Yaskawa INFORM job: DPRINT3D18.JBI

/JOB
//NAME DPRINT3D18
//POS
///NPOS 625,0,0,0,0,0
///TOOL 9
///POSTYPE PULSE
///PULSE
C00000=36096,32575,-120643,81709,-123035,-81395,0
C00001=36425,32776,-120243,81467,-123331,-81351,0
C00002=34958,34612,-116515,83246,-122769,-80325,0
C00003=34636,34416,-116909,83476,-122474,-80372,0
C00004=34349,34800,-116126,83824,-122361,-80159,0
C00005=35252,35359,-115002,83189,-123196,-80022,0
C00006=35016,35676,-114352,83478,-123103,-79844,0
C00007=35485,35977,-113744,83156,-123545,-79768,0
C00008=35668,35733,-114245,82930,-123616,-79906,0
C00009=36231,35313,-115109,82324,-123921,-80177,0
C00010=38030,32425,-120969,79919,-124380,-81738,0
C00011=40285,30090,-125653,77187,-125198,-83094,0
C00012=40286,30038,-125645,77208,-125225,-83061,0
C00013=36418,35187,-115263,82157,-124059,-80209,0
C00014=41098,30074,-125584,76447,-125785,-83178,0
C00015=40091,29408,-126885,77224,-124886,-83293,0
C00016=37256,32373,-120954,80642,-123847,-81594,0
C00017=37581,32580,-120545,80403,-124142,-81550,0
C00018=35772,34768,-116105,82607,-123455,-80311,0
C00019=36340,35136,-115366,82211,-123986,-80222,0
C00020=35723,35614,-114384,82881,-123656,-79916,0
C00021=36597,36197,-113208,82288,-124488,-79769,0
C00022=47213,22031,-141100,88472,-114439,-84668,0
C00023=39961,28432,-128797,77096,-124480,-83674,0
C00024=36097,32526,-120634,81728,-123056,-81363,0
C00025=36425,32727,-120235,81485,-123353,-81319,0
C00026=34959,34565,-116507,83263,-122787,-80294,0
C00027=34636,34368,-116901,83493,-122492,-80341,0
C00028=34350,34753,-116118,83841,-122379,-80128,0
C00029=35253,35312,-114994,83206,-123215,-79992,0
C00030=35016,35630,-114344,83496,-123122,-79813,0
C00031=35485,35931,-113736,83174,-123563,-79737,0
C00032=35669,35686,-114237,82948,-123634,-79875,0
C00033=36231,35266,-115101,82343,-123941,-80147,0
C00034=38031,32375,-120961,79938,-124402,-81706,0
C00035=40286,30038,-125645,77208,-125225,-83061,0
C00036=40286,29986,-125636,77229,-125250,-83028,0
C00037=36419,35140,-115255,82176,-124079,-80178,0
C00038=41098,30022,-125576,76469,-125813,-83145,0
C00039=40091,29355,-126877,77245,-124912,-83260,0
C00040=37256,32324,-120946,80661,-123870,-81562,0
C00041=37581,32531,-120536,80423,-124165,-81518,0
C00042=35772,34721,-116097,82625,-123474,-80280,0
C00043=36341,35089,-115358,82229,-124005,-80191,0
C00044=35723,35568,-114376,82899,-123674,-79885,0
C00045=36598,36150,-113200,82307,-124508,-79739,0
C00046=47214,21968,-141090,88484,-114457,-84628,0
C00047=39961,28378,-128788,77117,-124508,-83641,0
C00048=36097,32476,-120626,81746,-123078,-81331,0
C00049=36425,32677,-120226,81504,-123373,-81287,0
C00050=34959,34517,-116499,83281,-122807,-80263,0
C00051=34636,34320,-116893,83511,-122511,-80310,0
C00052=34350,34705,-116110,83858,-122398,-80098,0
C00053=35253,35265,-114985,83224,-123233,-79961,0
C00054=35016,35583,-114335,83514,-123140,-79783,0
C00055=35485,35885,-113727,83192,-123581,-79707,0
C00056=35669,35640,-114229,82966,-123654,-79845,0
C00057=36231,35219,-115093,82361,-123961,-80116,0
C00058=38031,32326,-120953,79958,-124425,-81674,0
C00059=40286,29986,-125636,77229,-125250,-83028,0
C00060=40286,29934,-125628,77250,-125276,-82995,0
C00061=36419,35093,-115247,82194,-124100,-80148,0
C00062=41099,29970,-125567,76490,-125839,-83112,0
C00063=40092,29302,-126868,77266,-124938,-83226,0
C00064=37257,32274,-120938,80680,-123892,-81529,0
C00065=37581,32481,-120528,80442,-124187,-81486,0
C00066=35773,34674,-116088,82643,-123493,-80249,0
C00067=36341,35042,-115350,82248,-124025,-80160,0
C00068=35724,35521,-114368,82917,-123694,-79855,0
C00069=36598,36104,-113191,82326,-124527,-79708,0
C00070=47215,21905,-141081,88497,-114476,-84588,0
C00071=39961,28324,-128780,77137,-124535,-83607,0
C00072=36097,32426,-120618,81764,-123099,-81299,0
C00073=36426,32628,-120218,81522,-123395,-81255,0
C00074=34959,34470,-116490,83298,-122825,-80232,0
C00075=34637,34273,-116885,83528,-122530,-80279,0
C00076=34350,34658,-116101,83875,-122416,-80067,0
C00077=35253,35218,-114976,83242,-123252,-79930,0
C00078=35017,35536,-114327,83531,-123158,-79752,0
C00079=35486,35838,-113719,83210,-123600,-79676,0
C00080=35669,35593,-114221,82984,-123672,-79815,0
C00081=36232,35172,-115084,82379,-123980,-80086,0
C00082=38031,32276,-120944,79978,-124448,-81642,0
C00083=40286,29934,-125628,77250,-125276,-82995,0
C00084=40287,29882,-125619,77271,-125303,-82962,0
C00085=36419,35046,-115237,82213,-124119,-80117,0
C00086=41099,29918,-125559,76511,-125867,-83079,0
C00087=40092,29249,-126859,77287,-124965,-83193,0
C00088=37257,32224,-120929,80700,-123913,-81497,0
C00089=37582,32432,-120519,80461,-124209,-81454,0
C00090=35773,34626,-116080,82661,-123512,-80218,0
C00091=36341,34995,-115341,82266,-124046,-80130,0
C00092=35724,35475,-114359,82935,-123712,-79824,0
C00093=36598,36058,-113183,82344,-124545,-79678,0
C00094=47215,21842,-141070,88510,-114494,-84548,0
C00095=39962,28270,-128771,77158,-124562,-83572,0
C00096=36098,32377,-120608,81783,-123119,-81266,0
C00097=36426,32579,-120209,81541,-123416,-81223,0
C00098=34960,34422,-116482,83316,-122845,-80201,0
C00099=34637,34225,-116876,83545,-122548,-80247,0
C00100=34351,34611,-116092,83892,-122434,-80036,0
C00101=35254,35172,-114968,83259,-123270,-79899,0
C00102=35017,35490,-114319,83549,-123177,-79722,0
C00103=35486,35792,-113711,83228,-123618,-79646,0
C00104=35670,35547,-114212,83002,-123691,-79784,0
C00105=36232,35125,-115075,82398,-124000,-80055,0
C00106=38032,32226,-120936,79997,-124471,-81610,0
C00107=40287,29882,-125619,77271,-125303,-82962,0
C00108=40287,29829,-125610,77292,-125329,-82929,0
C00109=36419,34999,-115229,82231,-124139,-80087,0
C00110=41100,29866,-125550,76533,-125893,-83046,0
C00111=40093,29196,-126850,77308,-124991,-83160,0
C00112=37257,32175,-120920,80719,-123935,-81465,0
C00113=37582,32382,-120511,80480,-124232,-81422,0
C00114=35773,34579,-116072,82680,-123532,-80187,0
C00115=36342,34948,-115333,82285,-124065,-80099,0
C00116=35724,35428,-114351,82953,-123731,-79794,0
C00117=36599,36012,-113174,82363,-124565,-79648,0
C00118=47216,21778,-141061,88523,-114513,-84508,0
C00119=39962,28216,-128762,77179,-124589,-83539,0
C00120=36098,32328,-120600,81801,-123140,-81234,0
C00121=36427,32530,-120201,81559,-123437,-81191,0
C00122=34960,34375,-116474,83334,-122863,-80170,0
C00123=34638,34177,-116868,83563,-122567,-80217,0
C00124=34351,34564,-116084,83910,-122453,-80005,0
C00125=35254,35125,-114959,83277,-123289,-79868,0
C00126=35018,35444,-114310,83566,-123195,-79692,0
C00127=35487,35746,-113702,83246,-123636,-79615,0
C00128=35670,35500,-114204,83020,-123710,-79754,0
C00129=36232,35078,-115067,82416,-124019,-80024,0
C00130=38032,32177,-120927,80017,-124493,-81579,0
C00131=40287,29829,-125610,77292,-125329,-82929,0
C00132=40288,29777,-125600,77313,-125356,-82895,0
C00133=36420,34953,-115220,82250,-124158,-80056,0
C00134=41100,29814,-125541,76555,-125921,-83013,0
C00135=40093,29143,-126841,77329,-125019,-83126,0
C00136=37258,32125,-120912,80738,-123957,-81433,0
C00137=37583,32333,-120502,80500,-124254,-81390,0
C00138=35774,34532,-116062,82698,-123551,-80156,0
C00139=36342,34901,-115324,82303,-124085,-80068,0
C00140=35725,35382,-114342,82972,-123750,-79763,0
C00141=36599,35967,-113166,82382,-124585,-79617,0
C00142=47216,21715,-141051,88536,-114531,-84467,0
C00143=39963,28162,-128753,77200,-124617,-83504,0
C00144=36098,32278,-120591,81820,-123162,-81203,0
C00145=36427,32481,-120191,81578,-123458,-81160,0
C00146=34960,34327,-116465,83351,-122882,-80139,0
C00147=34638,34130,-116859,83580,-122586,-80185,0
C00148=34351,34516,-116075,83927,-122471,-79974,0
C00149=35254,35078,-114951,83295,-123308,-79838,0
C00150=35018,35397,-114302,83584,-123214,-79661,0
C00151=35487,35700,-113694,83264,-123655,-79585,0
C00152=35670,35454,-114195,83038,-123728,-79723,0
C00153=36233,35031,-115058,82435,-124039,-79993,0
C00154=38033,32127,-120919,80037,-124516,-81547,0
C00155=40288,29777,-125600,77313,-125356,-82895,0
C00156=40288,29725,-125592,77334,-125382,-82862,0
C00157=36420,34906,-115212,82268,-124178,-80025,0
C00158=41101,29762,-125531,76576,-125947,-82980,0
C00159=40093,29091,-126832,77350,-125045,-83092,0
C00160=37258,32076,-120903,80757,-123979,-81401,0
C00161=37583,32284,-120492,80519,-124275,-81358,0
C00162=35774,34485,-116053,82716,-123571,-80125,0
C00163=36342,34854,-115315,82322,-124104,-80037,0
C00164=35725,35335,-114333,82990,-123769,-79733,0
C00165=36599,35921,-113157,82400,-124603,-79587,0
C00166=47217,21652,-141040,88549,-114550,-84427,0
C00167=39963,28108,-128743,77221,-124644,-83470,0
C00168=36099,32229,-120582,81838,-123183,-81171,0
C00169=36427,32431,-120183,81597,-123479,-81128,0
C00170=34961,34280,-116457,83369,-122901,-80108,0
C00171=34638,34082,-116851,83598,-122605,-80154,0
C00172=34352,34469,-116067,83944,-122490,-79943,0
C00173=35254,35031,-114942,83313,-123326,-79807,0
C00174=35018,35351,-114293,83602,-123231,-79630,0
C00175=35487,35654,-113685,83282,-123673,-79555,0
C00176=35671,35407,-114186,83056,-123747,-79692,0
C00177=36233,34985,-115050,82453,-124058,-79962,0
C00178=38033,32078,-120910,80056,-124539,-81514,0
C00179=40288,29725,-125592,77334,-125382,-82862,0
C00180=40288,29673,-125583,77356,-125408,-82829,0
C00181=36421,34859,-115203,82287,-124197,-79994,0
C00182=41101,29710,-125522,76598,-125975,-82947,0
C00183=40094,29038,-126823,77371,-125072,-83059,0
C00184=37258,32026,-120893,80776,-124001,-81369,0
C00185=37583,32234,-120484,80539,-124297,-81326,0
C00186=35774,34438,-116045,82734,-123591,-80094,0
C00187=36342,34808,-115306,82341,-124124,-80007,0
C00188=35725,35289,-114325,83008,-123787,-79702,0
C00189=36600,35875,-113149,82419,-124622,-79557,0
C00190=47217,21590,-141030,88562,-114568,-84386,0
C00191=39963,28054,-128734,77242,-124671,-83436,0
C00192=36099,32180,-120574,81857,-123203,-81138,0
C00193=36428,32382,-120174,81615,-123500,-81096,0
C00194=34961,34233,-116447,83387,-122919,-80077,0
C00195=34639,34035,-116842,83615,-122623,-80123,0
C00196=34352,34422,-116058,83961,-122507,-79912,0
C00197=35255,34985,-114934,83331,-123345,-79776,0
C00198=35018,35304,-114284,83619,-123249,-79599,0
C00199=35487,35608,-113676,83300,-123692,-79524,0
C00200=35671,35361,-114178,83075,-123765,-79662,0
C00201=36233,34938,-115041,82472,-124078,-79932,0
C00202=38033,32028,-120900,80076,-124562,-81482,0
C00203=40288,29673,-125583,77356,-125408,-82829,0
C00204=40289,29621,-125574,77377,-125435,-82796,0
C00205=36421,34812,-115195,82306,-124217,-79963,0
C00206=41101,29658,-125513,76620,-126001,-82914,0
C00207=40094,28985,-126814,77392,-125098,-83025,0
C00208=37259,31977,-120884,80796,-124024,-81337,0
C00209=37584,32185,-120475,80558,-124320,-81294,0
C00210=35775,34391,-116036,82752,-123609,-80063,0
C00211=36343,34761,-115297,82359,-124143,-79976,0
C00212=35726,35243,-114316,83026,-123807,-79671,0
C00213=36600,35829,-113140,82438,-124641,-79526,0
C00214=47218,21527,-141020,88574,-114586,-84346,0
C00215=39964,28000,-128725,77264,-124698,-83402,0
C00216=36099,32130,-120565,81875,-123224,-81106,0
C00217=36428,32333,-120165,81634,-123522,-81064,0
C00218=34961,34186,-116438,83404,-122938,-80045,0
C00219=34639,33987,-116832,83633,-122641,-80092,0
C00220=34352,34375,-116049,83979,-122525,-79881,0
C00221=35255,34938,-114925,83349,-123363,-79745,0
C00222=35019,35258,-114275,83637,-123268,-79569,0
C00223=35488,35562,-113667,83318,-123710,-79494,0
C00224=35671,35315,-114169,83093,-123785,-79631,0
C00225=36234,34891,-115032,82490,-124096,-79901,0
C00226=38034,31979,-120891,80096,-124583,-81450,0
C00227=40289,29621,-125574,77377,-125435,-82796,0
C00228=40289,29570,-125564,77398,-125461,-82763,0
C00229=36421,34766,-115186,82324,-124236,-79932,0
C00230=41102,29606,-125504,76641,-126029,-82881,0
C00231=40095,28933,-126804,77413,-125125,-82991,0
C00232=35457,34141,-116430,82993,-123333,-80080,0
C00233=36343,34714,-115289,82378,-124163,-79944,0
C00234=35726,35196,-114307,83044,-123825,-79641,0
C00235=36600,35783,-113131,82457,-124660,-79496,0
C00236=47218,21464,-141009,88587,-114605,-84306,0
C00237=39964,27947,-128715,77285,-124726,-83367,0
C00238=34353,34328,-116041,83996,-122544,-79850,0
C00239=35256,34892,-114916,83367,-123383,-79715,0
C00240=35019,35212,-114266,83655,-123286,-79538,0
C00241=35488,35516,-113658,83336,-123728,-79463,0
C00242=35672,35269,-114160,83111,-123803,-79600,0
C00243=36234,34845,-115024,82509,-124116,-79870,0
C00244=36199,34122,-116480,82342,-123887,-80190,0
C00245=40289,29570,-125564,77398,-125461,-82763,0
C00246=40290,29518,-125554,77419,-125488,-82729,0
C00247=36422,34719,-115176,82343,-124256,-79902,0
C00248=41102,29554,-125495,76663,-126055,-82847,0
C00249=40095,28880,-126794,77435,-125151,-82958,0
C00250=35457,34094,-116421,83011,-123352,-80048,0
C00251=36344,34667,-115280,82397,-124182,-79914,0
C00252=35726,35150,-114298,83063,-123843,-79610,0
C00253=36601,35738,-113122,82475,-124680,-79466,0
C00254=47219,21401,-140999,88600,-114623,-84266,0
C00255=39965,27893,-128705,77306,-124753,-83333,0
C00256=34353,34281,-116031,84013,-122562,-79819,0
C00257=35256,34845,-114907,83385,-123401,-79684,0
C00258=35019,35166,-114257,83673,-123304,-79508,0
C00259=35488,35470,-113649,83354,-123747,-79433,0
C00260=35672,35223,-114151,83129,-123822,-79570,0
C00261=36234,34798,-115014,82527,-124135,-79839,0
C00262=36199,34074,-116470,82360,-123907,-80159,0
C00263=40290,29518,-125554,77419,-125488,-82729,0
C00264=40290,29466,-125545,77441,-125513,-82696,0
C00265=36422,34673,-115167,82362,-124275,-79871,0
C00266=41103,29503,-125485,76685,-126083,-82814,0
C00267=40095,28828,-126785,77456,-125178,-82924,0
C00268=35458,34047,-116413,83030,-123371,-80017,0
C00269=36344,34621,-115271,82415,-124202,-79883,0
C00270=35727,35104,-114289,83081,-123863,-79580,0
C00271=36601,35692,-113113,82494,-124698,-79435,0
C00272=47220,21338,-140988,88614,-114642,-84225,0
C00273=39965,27839,-128696,77327,-124780,-83299,0
C00274=34353,34234,-116022,84031,-122580,-79787,0
C00275=35256,34799,-114898,83403,-123419,-79653,0
C00276=35020,35120,-114248,83691,-123323,-79477,0
C00277=35489,35424,-113640,83372,-123766,-79402,0
C00278=35672,35177,-114142,83147,-123841,-79539,0
C00279=36235,34752,-115005,82546,-124155,-79809,0
C00280=36200,34027,-116461,82379,-123927,-80128,0
C00281=40290,29466,-125545,77441,-125513,-82696,0
C00282=40291,29414,-125536,77462,-125539,-82662,0
C00283=36422,34626,-115158,82381,-124295,-79839,0
C00284=41103,29451,-125475,76707,-126109,-82781,0
C00285=40096,28775,-126775,77477,-125205,-82891,0
C00286=35458,34000,-116403,83048,-123391,-79986,0
C00287=36344,34574,-115261,82434,-124221,-79852,0
C00288=35727,35058,-114280,83099,-123881,-79549,0
C00289=36601,35646,-113104,82513,-124718,-79405,0
C00290=47220,21276,-140977,88627,-114660,-84185,0
C00291=39966,27786,-128686,77349,-124807,-83265,0
C00292=34354,34187,-116013,84048,-122599,-79756,0
C00293=35256,34753,-114889,83421,-123438,-79622,0
C00294=35020,35074,-114239,83709,-123341,-79446,0
C00295=35489,35378,-113631,83390,-123785,-79371,0
C00296=35673,35131,-114133,83166,-123859,-79509,0
C00297=36235,34706,-114996,82565,-124174,-79778,0
C00298=36200,33980,-116452,82398,-123947,-80097,0
C00299=40291,29414,-125536,77462,-125539,-82662,0
C00300=40291,29363,-125526,77484,-125566,-82629,0
C00301=36423,34580,-115149,82400,-124314,-79809,0
C00302=41103,29399,-125466,76729,-126137,-82748,0
C00303=40096,28723,-126766,77498,-125232,-82857,0
C00304=35458,33953,-116393,83066,-123409,-79955,0
C00305=36345,34528,-115252,82453,-124241,-79821,0
C00306=35727,35012,-114270,83118,-123900,-79518,0
C00307=36602,35601,-113094,82532,-124737,-79374,0
C00308=47221,21213,-140967,88640,-114679,-84144,0
C00309=39966,27732,-128677,77370,-124835,-83231,0
C00310=34354,34140,-116004,84066,-122616,-79725,0
C00311=35257,34706,-114879,83439,-123456,-79591,0
C00312=35020,35028,-114230,83726,-123360,-79415,0
C00313=35489,35332,-113622,83408,-123803,-79341,0
C00314=35673,35084,-114123,83184,-123878,-79478,0
C00315=36235,34659,-114987,82583,-124194,-79747,0
C00316=36200,33933,-116443,82416,-123966,-80065,0
C00317=40291,29363,-125526,77484,-125566,-82629,0
C00318=40291,29311,-125517,77505,-125592,-82596,0
C00319=36423,34533,-115140,82418,-124334,-79778,0
C00320=41104,29348,-125457,76751,-126163,-82714,0
C00321=40097,28671,-126755,77520,-125258,-82823,0
C00322=35459,33906,-116384,83084,-123428,-79924,0
C00323=36345,34481,-115243,82472,-124259,-79790,0
C00324=35728,34966,-114261,83136,-123919,-79487,0
C00325=36602,35555,-113085,82551,-124756,-79343,0
C00326=47221,21151,-140955,88653,-114697,-84104,0
C00327=39966,27679,-128666,77391,-124863,-83196,0
C00328=34354,34094,-115995,84083,-122634,-79694,0
C00329=35257,34660,-114870,83457,-123474,-79560,0
C00330=35021,34981,-114221,83744,-123377,-79385,0
C00331=35490,35286,-113613,83427,-123822,-79310,0
C00332=35673,35039,-114114,83202,-123896,-79447,0
C00333=36236,34613,-114978,82602,-124213,-79716,0
C00334=36201,33886,-116432,82435,-123986,-80034,0
C00335=40291,29311,-125517,77505,-125592,-82596,0
C00336=40292,29259,-125506,77527,-125619,-82563,0
C00337=36423,34487,-115130,82437,-124354,-79747,0
C00338=41104,29296,-125446,76773,-126190,-82681,0
C00339=40097,28618,-126746,77541,-125284,-82790,0
C00340=35459,33859,-116375,83102,-123448,-79892,0
C00341=36345,34435,-115233,82491,-124279,-79759,0
C00342=35728,34920,-114252,83155,-123938,-79456,0
C00343=36602,35510,-113076,82570,-124775,-79313,0
C00344=47222,21088,-140945,88666,-114715,-84063,0
C00345=39967,27625,-128656,77413,-124889,-83162,0
C00346=34354,34047,-115984,84101,-122653,-79662,0
C00347=35257,34614,-114861,83475,-123494,-79530,0
C00348=35021,34936,-114211,83762,-123395,-79354,0
C00349=35490,35241,-113603,83445,-123840,-79280,0
C00350=35674,34993,-114105,83221,-123916,-79416,0
C00351=36236,34567,-114968,82621,-124232,-79685,0
C00352=36201,33839,-116423,82454,-124005,-80003,0
C00353=40292,29259,-125506,77527,-125619,-82563,0
C00354=40292,29208,-125497,77548,-125645,-82529,0
C00355=36424,34441,-115120,82456,-124373,-79716,0
C00356=41105,29245,-125436,76795,-126218,-82647,0
C00357=40097,28566,-126736,77563,-125311,-82756,0
C00358=35459,33812,-116366,83121,-123466,-79861,0
C00359=36346,34389,-115224,82509,-124298,-79728,0
C00360=35728,34874,-114242,83173,-123956,-79426,0
C00361=36603,35464,-113066,82589,-124794,-79282,0
C00362=47222,21026,-140934,88679,-114734,-84023,0
C00363=39967,27572,-128647,77434,-124917,-83128,0
C00364=34355,34000,-115975,84118,-122671,-79632,0
C00365=35258,34567,-114851,83493,-123512,-79498,0
C00366=35021,34890,-114202,83780,-123414,-79323,0
C00367=35490,35195,-113594,83463,-123858,-79249,0
C00368=35674,34947,-114095,83239,-123934,-79386,0
C00369=36236,34520,-114958,82640,-124251,-79654,0
C00370=36201,33792,-116414,82473,-124025,-79972,0
C00371=40292,29208,-125497,77548,-125645,-82529,0
C00372=40293,29157,-125487,77570,-125671,-82496,0
C00373=36424,34394,-115111,82475,-124393,-79685,0
C00374=41105,29193,-125427,76817,-126244,-82614,0
C00375=40098,28514,-126725,77584,-125337,-82722,0
C00376=35459,33765,-116355,83139,-123486,-79830,0
C00377=36346,34342,-115214,82528,-124318,-79697,0
C00378=35729,34828,-114233,83192,-123975,-79394,0
C00379=36603,35419,-113057,82608,-124813,-79252,0
C00380=47223,20964,-140922,88692,-114752,-83983,0
C00381=39968,27519,-128636,77456,-124944,-83093,0
C00382=34355,33954,-115966,84136,-122690,-79600,0
C00383=35258,34521,-114841,83511,-123531,-79468,0
C00384=35022,34844,-114192,83798,-123432,-79292,0
C00385=35491,35150,-113584,83482,-123877,-79218,0
C00386=35674,34901,-114086,83258,-123953,-79354,0
C00387=36237,34474,-114949,82659,-124271,-79623,0
C00388=36202,33746,-116405,82491,-124046,-79940,0
C00389=40293,29157,-125487,77570,-125671,-82496,0
C00390=40293,29105,-125476,77591,-125697,-82462,0
C00391=36424,34348,-115102,82494,-124412,-79654,0
C00392=41106,29142,-125417,76839,-126272,-82581,0
C00393=40098,28462,-126716,77606,-125364,-82688,0
C00394=35460,33718,-116346,83157,-123504,-79798,0
C00395=36346,34296,-115204,82547,-124337,-79666,0
C00396=35729,34782,-114223,83210,-123994,-79364,0
C00397=36603,35374,-113047,82627,-124833,-79221,0
C00398=47224,20901,-140911,88706,-114771,-83942,0
C00399=39968,27466,-128626,77477,-124971,-83059,0
C00400=34356,33907,-115956,84154,-122707,-79569,0
C00401=35258,34475,-114832,83529,-123549,-79437,0
C00402=35022,34798,-114182,83816,-123450,-79261,0
C00403=35491,35104,-113575,83500,-123895,-79187,0
C00404=35675,34855,-114076,83276,-123971,-79324,0
C00405=36237,34428,-114939,82677,-124290,-79592,0
C00406=36202,33699,-116395,82510,-124065,-79909,0
C00407=40293,29105,-125476,77591,-125697,-82462,0
C00408=40293,29054,-125466,77613,-125723,-82429,0
C00409=36425,34302,-115091,82513,-124432,-79623,0
C00410=41106,29091,-125406,76861,-126298,-82548,0
C00411=40099,28410,-126706,77628,-125390,-82654,0
C00412=35460,33672,-116336,83176,-123524,-79767,0
C00413=36347,34250,-115195,82566,-124357,-79635,0
C00414=35729,34736,-114213,83229,-124012,-79333,0
C00415=36604,35328,-113037,82646,-124851,-79191,0
C00416=47224,20839,-140899,88719,-114789,-83901,0
C00417=39969,27412,-128616,77499,-124998,-83025,0
C00418=34356,33860,-115946,84171,-122725,-79538,0
C00419=35259,34429,-114822,83548,-123568,-79405,0
C00420=35022,34752,-114173,83834,-123469,-79230,0
C00421=35491,35058,-113565,83518,-123913,-79156,0
C00422=35675,34809,-114066,83295,-123989,-79293,0
C00423=36237,34382,-114929,82696,-124310,-79561,0
C00424=36202,33652,-116385,82529,-124085,-79878,0
C00425=40293,29054,-125466,77613,-125723,-82429,0
C00426=40294,29002,-125456,77635,-125750,-82396,0
C00427=36425,34256,-115081,82532,-124451,-79592,0
C00428=41106,29039,-125396,76883,-126326,-82514,0
C00429=40099,28358,-126696,77649,-125417,-82620,0
C00430=35461,33625,-116327,83194,-123543,-79736,0
C00431=36347,34204,-115184,82585,-124377,-79604,0
C00432=35730,34691,-114203,83247,-124031,-79302,0
C00433=36604,35283,-113028,82666,-124871,-79160,0
C00434=47225,20777,-140888,88732,-114807,-83861,0
C00435=39969,27359,-128605,77520,-125026,-82990,0
C00436=34356,33814,-115936,84189,-122744,-79506,0
C00437=35259,34383,-114812,83566,-123586,-79375,0
C00438=35023,34706,-114163,83853,-123486,-79199,0
C00439=35492,35013,-113555,83537,-123931,-79126,0
C00440=35675,34764,-114057,83313,-124009,-79262,0
C00441=36238,34336,-114919,82715,-124328,-79530,0
C00442=36203,33605,-116375,82548,-124104,-79846,0
C00443=40294,29002,-125456,77635,-125750,-82396,0
C00444=40294,28951,-125445,77656,-125776,-82362,0
C00445=36425,34210,-115072,82551,-124471,-79560,0
C00446=41107,28988,-125386,76906,-126352,-82481,0
C00447=40100,28306,-126685,77671,-125443,-82586,0
C00448=35461,33578,-116316,83213,-123562,-79704,0
C00449=36347,34157,-115175,82604,-124396,-79573,0
C00450=35730,34645,-114194,83266,-124050,-79271,0
C00451=36604,35238,-113018,82685,-124889,-79129,0
C00452=47225,20715,-140876,88746,-114826,-83820,0
C00453=39969,27306,-128595,77542,-125052,-82956,0
C00454=34356,33767,-115927,84207,-122762,-79475,0
C00455=35259,34337,-114802,83584,-123604,-79343,0
C00456=35023,34661,-114153,83871,-123504,-79169,0
C00457=35492,34968,-113545,83555,-123949,-79095,0
C00458=35676,34718,-114047,83332,-124027,-79231,0
C00459=36238,34290,-114910,82734,-124348,-79499,0
C00460=36203,33559,-116365,82567,-124124,-79815,0
C00461=40294,28951,-125445,77656,-125776,-82362,0
C00462=40295,28900,-125435,77678,-125802,-82328,0
C00463=36426,34164,-115061,82571,-124490,-79530,0
C00464=41107,28937,-125375,76928,-126378,-82447,0
C00465=40100,28254,-126675,77693,-125469,-82553,0
C00466=35461,33532,-116306,83231,-123581,-79672,0
C00467=36348,34111,-115165,82623,-124416,-79541,0
C00468=35730,34599,-114184,83284,-124069,-79240,0
C00469=36605,35193,-113008,82704,-124909,-79098,0
C00470=47226,20653,-140865,88759,-114844,-83779,0
C00471=39970,27253,-128584,77564,-125080,-82921,0
C00472=34357,33721,-115916,84224,-122780,-79444,0
C00473=35260,34291,-114792,83603,-123623,-79313,0
C00474=35023,34615,-114143,83889,-123523,-79137,0
C00475=35492,34922,-113535,83574,-123967,-79064,0
C00476=35676,34673,-114037,83350,-124046,-79200,0
C00477=36238,34244,-114900,82753,-124367,-79468,0
C00478=36203,33512,-116355,82586,-124143,-79783,0
C00479=40295,28900,-125435,77678,-125802,-82328,0
C00480=40295,28849,-125425,77700,-125828,-82295,0
C00481=36426,34118,-115051,82590,-124510,-79498,0
C00482=41108,28886,-125365,76950,-126406,-82414,0
C00483=40100,28202,-126663,77714,-125497,-82519,0
C00484=35462,33485,-116297,83250,-123600,-79641,0
C00485=36348,34065,-115155,82642,-124435,-79510,0
C00486=35731,34554,-114174,83303,-124087,-79209,0
C00487=36605,35148,-112998,82723,-124927,-79068,0
C00488=47226,20591,-140853,88772,-114862,-83739,0
C00489=39970,27200,-128573,77585,-125106,-82886,0
C00490=34357,33675,-115906,84242,-122798,-79412,0
C00491=35260,34245,-114782,83621,-123641,-79281,0
C00492=35024,34570,-114133,83907,-123541,-79107,0
C00493=35493,34877,-113525,83592,-123986,-79033,0
C00494=35676,34627,-114027,83369,-124064,-79169,0
C00495=36239,34198,-114889,82772,-124387,-79437,0
C00496=36204,33465,-116345,82605,-124163,-79752,0
C00497=40295,28849,-125425,77700,-125828,-82295,0
C00498=40295,28798,-125414,77722,-125854,-82261,0
C00499=36426,34072,-115042,82609,-124528,-79467,0
C00500=45731,20512,-140851,90157,-113886,-83584,0
C00501=40101,28150,-126653,77736,-125523,-82484,0
C00502=35462,33439,-116286,83268,-123619,-79610,0
C00503=36348,34019,-115144,82662,-124455,-79479,0
C00504=35731,34508,-114163,83322,-124107,-79178,0
C00505=36605,35103,-112988,82743,-124947,-79038,0
C00506=47227,20529,-140842,88786,-114881,-83698,0
C00507=39971,27147,-128563,77607,-125134,-82852,0
C00508=34357,33628,-115896,84260,-122816,-79381,0
C00509=35260,34200,-114772,83639,-123661,-79250,0
C00510=35024,34524,-114123,83925,-123558,-79076,0
C00511=35493,34832,-113515,83611,-124004,-79003,0
C00512=35677,34582,-114016,83388,-124082,-79139,0
C00513=36239,34152,-114879,82791,-124406,-79405,0
C00514=36204,33419,-116335,82624,-124183,-79721,0
C00515=40295,28798,-125414,77722,-125854,-82261,0
C00516=40296,28747,-125404,77744,-125881,-82227,0
C00517=36427,34026,-115032,82628,-124548,-79436,0
C00518=45732,20450,-140839,90169,-113903,-83543,0
C00519=40101,28098,-126643,77758,-125550,-82451,0
C00520=35462,33392,-116276,83287,-123639,-79578,0
C00521=36349,33973,-115134,82681,-124474,-79448,0
C00522=35731,34463,-114153,83340,-124125,-79147,0
C00523=36606,35058,-112978,82762,-124966,-79007,0
C00524=47227,20468,-140829,88799,-114899,-83658,0
C00525=39971,27094,-128551,77629,-125161,-82817,0
C00526=34358,33582,-115885,84278,-122834,-79350,0
C00527=35261,34154,-114762,83658,-123679,-79219,0
C00528=35024,34478,-114113,83943,-123577,-79045,0
C00529=35493,34786,-113505,83629,-124023,-78972,0
C00530=35677,34536,-114006,83406,-124102,-79107,0
C00531=36239,34106,-114869,82810,-124425,-79375,0
C00532=36204,33372,-116324,82643,-124203,-79689,0
C00533=40296,28747,-125404,77744,-125881,-82227,0
C00534=40296,28696,-125392,77766,-125906,-82194,0
C00535=36427,33980,-115021,82647,-124567,-79405,0
C00536=45733,20388,-140827,90181,-113919,-83502,0
C00537=40102,28047,-126631,77780,-125576,-82416,0
C00538=35463,33346,-116266,83306,-123657,-79546,0
C00539=36349,33927,-115124,82700,-124494,-79416,0
C00540=35732,34417,-114143,83359,-124143,-79116,0
C00541=36606,35013,-112967,82781,-124984,-78976,0
C00542=47228,20406,-140818,88813,-114917,-83617,0
C00543=39971,27041,-128541,77651,-125188,-82783,0
C00544=34358,33536,-115875,84296,-122853,-79318,0
C00545=35261,34108,-114751,83676,-123697,-79188,0
C00546=35025,34433,-114102,83962,-123595,-79014,0
C00547=35494,34741,-113495,83648,-124041,-78941,0
C00548=35677,34491,-113996,83425,-124120,-79076,0
C00549=36240,34060,-114859,82830,-124444,-79343,0
C00550=36205,33326,-116314,82662,-124223,-79657,0
C00551=40296,28696,-125392,77766,-125906,-82194,0
C00552=40297,28645,-125382,77788,-125933,-82160,0
C00553=36427,33934,-115011,82667,-124587,-79374,0
C00554=45733,20327,-140815,90194,-113936,-83461,0
C00555=40102,27995,-126621,77802,-125603,-82383,0
C00556=35463,33299,-116255,83324,-123677,-79515,0
C00557=36349,33882,-115113,82719,-124513,-79385,0
C00558=35732,34372,-114132,83378,-124162,-79085,0
C00559=36606,34968,-112957,82801,-125004,-78945,0
C00560=47229,20344,-140805,88826,-114935,-83576,0
C00561=39972,26988,-128530,77673,-125215,-82748,0
C00562=34358,33490,-115865,84313,-122870,-79286,0
C00563=35261,34062,-114741,83695,-123716,-79156,0
C00564=35025,34388,-114092,83980,-123614,-78982,0
C00565=35494,34696,-113484,83666,-124059,-78910,0
C00566=35678,34445,-113986,83444,-124139,-79046,0
C00567=36240,34015,-114848,82849,-124464,-79312,0
C00568=36205,33280,-116304,82682,-124242,-79626,0
C00569=40297,28645,-125382,77788,-125933,-82160,0
C00570=40297,28594,-125371,77810,-125959,-82126,0
C00571=36428,33888,-114999,82686,-124606,-79342,0
C00572=45734,20265,-140803,90206,-113953,-83421,0
C00573=40103,27943,-126609,77824,-125629,-82349,0
C00574=35463,33253,-116244,83343,-123695,-79484,0
C00575=36350,33836,-115103,82738,-124532,-79354,0
C00576=35732,34326,-114122,83397,-124181,-79054,0
C00577=36607,34923,-112946,82820,-125022,-78914,0
C00578=47229,20283,-140792,88840,-114953,-83536,0
C00579=39972,26936,-128518,77695,-125242,-82714,0
C00580=34359,33443,-115854,84331,-122888,-79255,0
C00581=35262,34017,-114731,83713,-123734,-79125,0
C00582=35025,34342,-114081,83998,-123632,-78952,0
C00583=35494,34651,-113474,83685,-124078,-78879,0
C00584=35678,34400,-113975,83463,-124157,-79014,0
C00585=36240,33969,-114838,82868,-124483,-79281,0
C00586=36205,33233,-116293,82701,-124262,-79595,0
C00587=40297,28594,-125371,77810,-125959,-82126,0
C00588=40297,28543,-125360,77832,-125985,-82093,0
C00589=36428,33843,-114989,82705,-124626,-79311,0
C00590=45734,20203,-140790,90218,-113969,-83380,0
C00591=40103,27892,-126598,77846,-125656,-82314,0
C00592=35464,33207,-116234,83362,-123715,-79452,0
C00593=36350,33790,-115093,82758,-124551,-79323,0
C00594=35732,34281,-114111,83416,-124200,-79023,0
C00595=36607,34878,-112936,82839,-125042,-78883,0
C00596=47230,20221,-140781,88853,-114972,-83495,0
C00597=39973,26883,-128508,77717,-125269,-82679,0
C00598=34359,33397,-115844,84349,-122907,-79224,0
C00599=35262,33971,-114720,83732,-123753,-79094,0
C00600=35026,34297,-114071,84017,-123649,-78920,0
C00601=35495,34606,-113463,83704,-124096,-78848,0
C00602=35678,34355,-113965,83481,-124175,-78984,0
C00603=36241,33923,-114827,82887,-124502,-79249,0
C00604=36206,33187,-116282,82720,-124281,-79563,0
C00605=40297,28543,-125360,77832,-125985,-82093,0
C00606=40298,28492,-125349,77854,-126011,-82059,0
C00607=36428,33797,-114979,82725,-124645,-79280,0
C00608=45735,20142,-140778,90231,-113986,-83339,0
C00609=40103,27840,-126588,77868,-125682,-82280,0
C00610=35464,33160,-116223,83380,-123734,-79421,0
C00611=36350,33744,-115082,82777,-124571,-79292,0
C00612=35733,34236,-114101,83435,-124218,-78992,0
C00613=36607,34833,-112925,82859,-125060,-78852,0
C00614=47230,20160,-140768,88867,-114990,-83455,0
C00615=39973,26830,-128496,77739,-125296,-82644,0
C00616=34359,33351,-115833,84367,-122924,-79192,0
C00617=35262,33926,-114709,83750,-123771,-79063,0
C00618=35026,34252,-114060,84035,-123668,-78889,0
C00619=35495,34561,-113453,83723,-124115,-78817,0
C00620=35679,34310,-113954,83500,-124194,-78952,0
C00621=36241,33878,-114817,82906,-124521,-79219,0
C00622=36206,33141,-116272,82739,-124301,-79531,0
C00623=40298,28492,-125349,77854,-126011,-82059,0
C00624=44783,17058,-140181,91723,-114080,-81234,0
//INST
///DATE 2025/02/20 16:20
///COMM Generated using RoboDK
///ATTR SC,RW
///GROUP1 RB1
NOP
MOVL C00000 V=30.0 PL=1
MOVL C00001 V=30.0 PL=1
MOVL C00002 V=30.0 PL=1
MOVL C00003 V=30.0 PL=1
MOVL C00004 V=30.0 PL=1
MOVL C00005 V=30.0 PL=1
MOVL C00006 V=30.0 PL=1
MOVL C00007 V=30.0 PL=1
MOVL C00008 V=30.0 PL=1
MOVL C00009 V=130.0 PL=1
MOVL C00010 V=130.0 PL=1
MOVL C00011 V=20.0 PL=1
MOVL C00012 V=130.0 PL=1
MOVL C00013 V=130.0 PL=1
MOVL C00014 V=60.0 PL=1
MOVL C00015 V=60.0 PL=1
MOVL C00016 V=60.0 PL=1
MOVL C00017 V=60.0 PL=1
MOVL C00018 V=60.0 PL=1
MOVL C00019 V=60.0 PL=1
MOVL C00020 V=130.0 PL=1
MOVL C00021 V=30.0 PL=1
MOVL C00022 V=30.0 PL=1
MOVL C00023 V=30.0 PL=1
MOVL C00024 V=30.0 PL=1
MOVL C00025 V=30.0 PL=1
MOVL C00026 V=30.0 PL=1
MOVL C00027 V=30.0 PL=1
MOVL C00028 V=30.0 PL=1
MOVL C00029 V=30.0 PL=1
MOVL C00030 V=30.0 PL=1
MOVL C00031 V=30.0 PL=1
MOVL C00032 V=30.0 PL=1
MOVL C00033 V=130.0 PL=1
MOVL C00034 V=130.0 PL=1
MOVL C00035 V=20.0 PL=1
MOVL C00036 V=130.0 PL=1
MOVL C00037 V=130.0 PL=1
MOVL C00038 V=60.0 PL=1
MOVL C00039 V=60.0 PL=1
MOVL C00040 V=60.0 PL=1
MOVL C00041 V=60.0 PL=1
MOVL C00042 V=60.0 PL=1
MOVL C00043 V=60.0 PL=1
MOVL C00044 V=130.0 PL=1
MOVL C00045 V=30.0 PL=1
MOVL C00046 V=30.0 PL=1
MOVL C00047 V=30.0 PL=1
MOVL C00048 V=30.0 PL=1
MOVL C00049 V=30.0 PL=1
MOVL C00050 V=30.0 PL=1
MOVL C00051 V=30.0 PL=1
MOVL C00052 V=30.0 PL=1
MOVL C00053 V=30.0 PL=1
MOVL C00054 V=30.0 PL=1
MOVL C00055 V=30.0 PL=1
MOVL C00056 V=30.0 PL=1
MOVL C00057 V=130.0 PL=1
MOVL C00058 V=130.0 PL=1
MOVL C00059 V=20.0 PL=1
MOVL C00060 V=130.0 PL=1
MOVL C00061 V=130.0 PL=1
MOVL C00062 V=60.0 PL=1
MOVL C00063 V=60.0 PL=1
MOVL C00064 V=60.0 PL=1
MOVL C00065 V=60.0 PL=1
MOVL C00066 V=60.0 PL=1
MOVL C00067 V=60.0 PL=1
MOVL C00068 V=130.0 PL=1
MOVL C00069 V=30.0 PL=1
MOVL C00070 V=30.0 PL=1
MOVL C00071 V=30.0 PL=1
MOVL C00072 V=30.0 PL=1
MOVL C00073 V=30.0 PL=1
MOVL C00074 V=30.0 PL=1
MOVL C00075 V=30.0 PL=1
MOVL C00076 V=30.0 PL=1
MOVL C00077 V=30.0 PL=1
MOVL C00078 V=30.0 PL=1
MOVL C00079 V=30.0 PL=1
MOVL C00080 V=30.0 PL=1
MOVL C00081 V=130.0 PL=1
MOVL C00082 V=130.0 PL=1
MOVL C00083 V=20.0 PL=1
MOVL C00084 V=130.0 PL=1
MOVL C00085 V=130.0 PL=1
MOVL C00086 V=60.0 PL=1
MOVL C00087 V=60.0 PL=1
MOVL C00088 V=60.0 PL=1
MOVL C00089 V=60.0 PL=1
MOVL C00090 V=60.0 PL=1
MOVL C00091 V=60.0 PL=1
MOVL C00092 V=130.0 PL=1
MOVL C00093 V=30.0 PL=1
MOVL C00094 V=30.0 PL=1
MOVL C00095 V=30.0 PL=1
MOVL C00096 V=30.0 PL=1
MOVL C00097 V=30.0 PL=1
MOVL C00098 V=30.0 PL=1
MOVL C00099 V=30.0 PL=1
MOVL C00100 V=30.0 PL=1
MOVL C00101 V=30.0 PL=1
MOVL C00102 V=30.0 PL=1
MOVL C00103 V=30.0 PL=1
MOVL C00104 V=30.0 PL=1
MOVL C00105 V=130.0 PL=1
MOVL C00106 V=130.0 PL=1
MOVL C00107 V=20.0 PL=1
MOVL C00108 V=130.0 PL=1
MOVL C00109 V=130.0 PL=1
MOVL C00110 V=60.0 PL=1
MOVL C00111 V=60.0 PL=1
MOVL C00112 V=60.0 PL=1
MOVL C00113 V=60.0 PL=1
MOVL C00114 V=60.0 PL=1
MOVL C00115 V=60.0 PL=1
MOVL C00116 V=130.0 PL=1
MOVL C00117 V=30.0 PL=1
MOVL C00118 V=30.0 PL=1
MOVL C00119 V=30.0 PL=1
MOVL C00120 V=30.0 PL=1
MOVL C00121 V=30.0 PL=1
MOVL C00122 V=30.0 PL=1
MOVL C00123 V=30.0 PL=1
MOVL C00124 V=30.0 PL=1
MOVL C00125 V=30.0 PL=1
MOVL C00126 V=30.0 PL=1
MOVL C00127 V=30.0 PL=1
MOVL C00128 V=30.0 PL=1
MOVL C00129 V=130.0 PL=1
MOVL C00130 V=130.0 PL=1
MOVL C00131 V=20.0 PL=1
MOVL C00132 V=130.0 PL=1
MOVL C00133 V=130.0 PL=1
MOVL C00134 V=60.0 PL=1
MOVL C00135 V=60.0 PL=1
MOVL C00136 V=60.0 PL=1
MOVL C00137 V=60.0 PL=1
MOVL C00138 V=60.0 PL=1
MOVL C00139 V=60.0 PL=1
MOVL C00140 V=130.0 PL=1
MOVL C00141 V=30.0 PL=1
MOVL C00142 V=30.0 PL=1
MOVL C00143 V=30.0 PL=1
MOVL C00144 V=30.0 PL=1
MOVL C00145 V=30.0 PL=1
MOVL C00146 V=30.0 PL=1
MOVL C00147 V=30.0 PL=1
MOVL C00148 V=30.0 PL=1
MOVL C00149 V=30.0 PL=1
MOVL C00150 V=30.0 PL=1
MOVL C00151 V=30.0 PL=1
MOVL C00152 V=30.0 PL=1
MOVL C00153 V=130.0 PL=1
MOVL C00154 V=130.0 PL=1
MOVL C00155 V=20.0 PL=1
MOVL C00156 V=130.0 PL=1
MOVL C00157 V=130.0 PL=1
MOVL C00158 V=60.0 PL=1
MOVL C00159 V=60.0 PL=1
MOVL C00160 V=60.0 PL=1
MOVL C00161 V=60.0 PL=1
MOVL C00162 V=60.0 PL=1
MOVL C00163 V=60.0 PL=1
MOVL C00164 V=130.0 PL=1
MOVL C00165 V=30.0 PL=1
MOVL C00166 V=30.0 PL=1
MOVL C00167 V=30.0 PL=1
MOVL C00168 V=30.0 PL=1
MOVL C00169 V=30.0 PL=1
MOVL C00170 V=30.0 PL=1
MOVL C00171 V=30.0 PL=1
MOVL C00172 V=30.0 PL=1
MOVL C00173 V=30.0 PL=1
MOVL C00174 V=30.0 PL=1
MOVL C00175 V=30.0 PL=1
MOVL C00176 V=30.0 PL=1
MOVL C00177 V=130.0 PL=1
MOVL C00178 V=130.0 PL=1
MOVL C00179 V=20.0 PL=1
MOVL C00180 V=130.0 PL=1
MOVL C00181 V=130.0 PL=1
MOVL C00182 V=60.0 PL=1
MOVL C00183 V=60.0 PL=1
MOVL C00184 V=60.0 PL=1
MOVL C00185 V=60.0 PL=1
MOVL C00186 V=60.0 PL=1
MOVL C00187 V=60.0 PL=1
MOVL C00188 V=130.0 PL=1
MOVL C00189 V=30.0 PL=1
MOVL C00190 V=30.0 PL=1
MOVL C00191 V=30.0 PL=1
MOVL C00192 V=30.0 PL=1
MOVL C00193 V=30.0 PL=1
MOVL C00194 V=30.0 PL=1
MOVL C00195 V=30.0 PL=1
MOVL C00196 V=30.0 PL=1
MOVL C00197 V=30.0 PL=1
MOVL C00198 V=30.0 PL=1
MOVL C00199 V=30.0 PL=1
MOVL C00200 V=30.0 PL=1
MOVL C00201 V=130.0 PL=1
MOVL C00202 V=130.0 PL=1
MOVL C00203 V=20.0 PL=1
MOVL C00204 V=130.0 PL=1
MOVL C00205 V=130.0 PL=1
MOVL C00206 V=60.0 PL=1
MOVL C00207 V=60.0 PL=1
MOVL C00208 V=60.0 PL=1
MOVL C00209 V=60.0 PL=1
MOVL C00210 V=60.0 PL=1
MOVL C00211 V=60.0 PL=1
MOVL C00212 V=130.0 PL=1
MOVL C00213 V=30.0 PL=1
MOVL C00214 V=30.0 PL=1
MOVL C00215 V=30.0 PL=1
MOVL C00216 V=30.0 PL=1
MOVL C00217 V=30.0 PL=1
MOVL C00218 V=30.0 PL=1
MOVL C00219 V=30.0 PL=1
MOVL C00220 V=30.0 PL=1
MOVL C00221 V=30.0 PL=1
MOVL C00222 V=30.0 PL=1
MOVL C00223 V=30.0 PL=1
MOVL C00224 V=30.0 PL=1
MOVL C00225 V=130.0 PL=1
MOVL C00226 V=130.0 PL=1
MOVL C00227 V=20.0 PL=1
MOVL C00228 V=130.0 PL=1
MOVL C00229 V=130.0 PL=1
MOVL C00230 V=60.0 PL=1
MOVL C00231 V=60.0 PL=1
MOVL C00232 V=60.0 PL=1
MOVL C00233 V=60.0 PL=1
MOVL C00234 V=130.0 PL=1
MOVL C00235 V=30.0 PL=1
MOVL C00236 V=30.0 PL=1
MOVL C00237 V=30.0 PL=1
MOVL C00238 V=30.0 PL=1
MOVL C00239 V=30.0 PL=1
MOVL C00240 V=30.0 PL=1
MOVL C00241 V=30.0 PL=1
MOVL C00242 V=30.0 PL=1
MOVL C00243 V=130.0 PL=1
MOVL C00244 V=130.0 PL=1
MOVL C00245 V=20.0 PL=1
MOVL C00246 V=130.0 PL=1
MOVL C00247 V=130.0 PL=1
MOVL C00248 V=60.0 PL=1
MOVL C00249 V=60.0 PL=1
MOVL C00250 V=60.0 PL=1
MOVL C00251 V=60.0 PL=1
MOVL C00252 V=130.0 PL=1
MOVL C00253 V=30.0 PL=1
MOVL C00254 V=30.0 PL=1
MOVL C00255 V=30.0 PL=1
MOVL C00256 V=30.0 PL=1
MOVL C00257 V=30.0 PL=1
MOVL C00258 V=30.0 PL=1
MOVL C00259 V=30.0 PL=1
MOVL C00260 V=30.0 PL=1
MOVL C00261 V=130.0 PL=1
MOVL C00262 V=130.0 PL=1
MOVL C00263 V=20.0 PL=1
MOVL C00264 V=130.0 PL=1
MOVL C00265 V=130.0 PL=1
MOVL C00266 V=60.0 PL=1
MOVL C00267 V=60.0 PL=1
MOVL C00268 V=60.0 PL=1
MOVL C00269 V=60.0 PL=1
MOVL C00270 V=130.0 PL=1
MOVL C00271 V=30.0 PL=1
MOVL C00272 V=30.0 PL=1
MOVL C00273 V=30.0 PL=1
MOVL C00274 V=30.0 PL=1
MOVL C00275 V=30.0 PL=1
MOVL C00276 V=30.0 PL=1
MOVL C00277 V=30.0 PL=1
MOVL C00278 V=30.0 PL=1
MOVL C00279 V=130.0 PL=1
MOVL C00280 V=130.0 PL=1
MOVL C00281 V=20.0 PL=1
MOVL C00282 V=130.0 PL=1
MOVL C00283 V=130.0 PL=1
MOVL C00284 V=60.0 PL=1
MOVL C00285 V=60.0 PL=1
MOVL C00286 V=60.0 PL=1
MOVL C00287 V=60.0 PL=1
MOVL C00288 V=130.0 PL=1
MOVL C00289 V=30.0 PL=1
MOVL C00290 V=30.0 PL=1
MOVL C00291 V=30.0 PL=1
MOVL C00292 V=30.0 PL=1
MOVL C00293 V=30.0 PL=1
MOVL C00294 V=30.0 PL=1
MOVL C00295 V=30.0 PL=1
MOVL C00296 V=30.0 PL=1
MOVL C00297 V=130.0 PL=1
MOVL C00298 V=130.0 PL=1
MOVL C00299 V=20.0 PL=1
MOVL C00300 V=130.0 PL=1
MOVL C00301 V=130.0 PL=1
MOVL C00302 V=60.0 PL=1
MOVL C00303 V=60.0 PL=1
MOVL C00304 V=60.0 PL=1
MOVL C00305 V=60.0 PL=1
MOVL C00306 V=130.0 PL=1
MOVL C00307 V=30.0 PL=1
MOVL C00308 V=30.0 PL=1
MOVL C00309 V=30.0 PL=1
MOVL C00310 V=30.0 PL=1
MOVL C00311 V=30.0 PL=1
MOVL C00312 V=30.0 PL=1
MOVL C00313 V=30.0 PL=1
MOVL C00314 V=30.0 PL=1
MOVL C00315 V=130.0 PL=1
MOVL C00316 V=130.0 PL=1
MOVL C00317 V=20.0 PL=1
MOVL C00318 V=130.0 PL=1
MOVL C00319 V=130.0 PL=1
MOVL C00320 V=60.0 PL=1
MOVL C00321 V=60.0 PL=1
MOVL C00322 V=60.0 PL=1
MOVL C00323 V=60.0 PL=1
MOVL C00324 V=130.0 PL=1
MOVL C00325 V=30.0 PL=1
MOVL C00326 V=30.0 PL=1
MOVL C00327 V=30.0 PL=1
MOVL C00328 V=30.0 PL=1
MOVL C00329 V=30.0 PL=1
MOVL C00330 V=30.0 PL=1
MOVL C00331 V=30.0 PL=1
MOVL C00332 V=30.0 PL=1
MOVL C00333 V=130.0 PL=1
MOVL C00334 V=130.0 PL=1
MOVL C00335 V=20.0 PL=1
MOVL C00336 V=130.0 PL=1
MOVL C00337 V=130.0 PL=1
MOVL C00338 V=60.0 PL=1
MOVL C00339 V=60.0 PL=1
MOVL C00340 V=60.0 PL=1
MOVL C00341 V=60.0 PL=1
MOVL C00342 V=130.0 PL=1
MOVL C00343 V=30.0 PL=1
MOVL C00344 V=30.0 PL=1
MOVL C00345 V=30.0 PL=1
MOVL C00346 V=30.0 PL=1
MOVL C00347 V=30.0 PL=1
MOVL C00348 V=30.0 PL=1
MOVL C00349 V=30.0 PL=1
MOVL C00350 V=30.0 PL=1
MOVL C00351 V=130.0 PL=1
MOVL C00352 V=130.0 PL=1
MOVL C00353 V=20.0 PL=1
MOVL C00354 V=130.0 PL=1
MOVL C00355 V=130.0 PL=1
MOVL C00356 V=60.0 PL=1
MOVL C00357 V=60.0 PL=1
MOVL C00358 V=60.0 PL=1
MOVL C00359 V=60.0 PL=1
MOVL C00360 V=130.0 PL=1
MOVL C00361 V=30.0 PL=1
MOVL C00362 V=30.0 PL=1
MOVL C00363 V=30.0 PL=1
MOVL C00364 V=30.0 PL=1
MOVL C00365 V=30.0 PL=1
MOVL C00366 V=30.0 PL=1
MOVL C00367 V=30.0 PL=1
MOVL C00368 V=30.0 PL=1
MOVL C00369 V=130.0 PL=1
MOVL C00370 V=130.0 PL=1
MOVL C00371 V=20.0 PL=1
MOVL C00372 V=130.0 PL=1
MOVL C00373 V=130.0 PL=1
MOVL C00374 V=60.0 PL=1
MOVL C00375 V=60.0 PL=1
MOVL C00376 V=60.0 PL=1
MOVL C00377 V=60.0 PL=1
MOVL C00378 V=130.0 PL=1
MOVL C00379 V=30.0 PL=1
MOVL C00380 V=30.0 PL=1
MOVL C00381 V=30.0 PL=1
MOVL C00382 V=30.0 PL=1
MOVL C00383 V=30.0 PL=1
MOVL C00384 V=30.0 PL=1
MOVL C00385 V=30.0 PL=1
MOVL C00386 V=30.0 PL=1
MOVL C00387 V=130.0 PL=1
MOVL C00388 V=130.0 PL=1
MOVL C00389 V=20.0 PL=1
MOVL C00390 V=130.0 PL=1
MOVL C00391 V=130.0 PL=1
MOVL C00392 V=60.0 PL=1
MOVL C00393 V=60.0 PL=1
MOVL C00394 V=60.0 PL=1
MOVL C00395 V=60.0 PL=1
MOVL C00396 V=130.0 PL=1
MOVL C00397 V=30.0 PL=1
MOVL C00398 V=30.0 PL=1
MOVL C00399 V=30.0 PL=1
MOVL C00400 V=30.0 PL=1
MOVL C00401 V=30.0 PL=1
MOVL C00402 V=30.0 PL=1
MOVL C00403 V=30.0 PL=1
MOVL C00404 V=30.0 PL=1
MOVL C00405 V=130.0 PL=1
MOVL C00406 V=130.0 PL=1
MOVL C00407 V=20.0 PL=1
MOVL C00408 V=130.0 PL=1
MOVL C00409 V=130.0 PL=1
MOVL C00410 V=60.0 PL=1
MOVL C00411 V=60.0 PL=1
MOVL C00412 V=60.0 PL=1
MOVL C00413 V=60.0 PL=1
MOVL C00414 V=130.0 PL=1
MOVL C00415 V=30.0 PL=1
MOVL C00416 V=30.0 PL=1
MOVL C00417 V=30.0 PL=1
MOVL C00418 V=30.0 PL=1
MOVL C00419 V=30.0 PL=1
MOVL C00420 V=30.0 PL=1
MOVL C00421 V=30.0 PL=1
MOVL C00422 V=30.0 PL=1
MOVL C00423 V=130.0 PL=1
MOVL C00424 V=130.0 PL=1
MOVL C00425 V=20.0 PL=1
MOVL C00426 V=130.0 PL=1
MOVL C00427 V=130.0 PL=1
MOVL C00428 V=60.0 PL=1
MOVL C00429 V=60.0 PL=1
MOVL C00430 V=60.0 PL=1
MOVL C00431 V=60.0 PL=1
MOVL C00432 V=130.0 PL=1
MOVL C00433 V=30.0 PL=1
MOVL C00434 V=30.0 PL=1
MOVL C00435 V=30.0 PL=1
MOVL C00436 V=30.0 PL=1
MOVL C00437 V=30.0 PL=1
MOVL C00438 V=30.0 PL=1
MOVL C00439 V=30.0 PL=1
MOVL C00440 V=30.0 PL=1
MOVL C00441 V=130.0 PL=1
MOVL C00442 V=130.0 PL=1
MOVL C00443 V=20.0 PL=1
MOVL C00444 V=130.0 PL=1
MOVL C00445 V=130.0 PL=1
MOVL C00446 V=60.0 PL=1
MOVL C00447 V=60.0 PL=1
MOVL C00448 V=60.0 PL=1
MOVL C00449 V=60.0 PL=1
MOVL C00450 V=130.0 PL=1
MOVL C00451 V=30.0 PL=1
MOVL C00452 V=30.0 PL=1
MOVL C00453 V=30.0 PL=1
MOVL C00454 V=30.0 PL=1
MOVL C00455 V=30.0 PL=1
MOVL C00456 V=30.0 PL=1
MOVL C00457 V=30.0 PL=1
MOVL C00458 V=30.0 PL=1
MOVL C00459 V=130.0 PL=1
MOVL C00460 V=130.0 PL=1
MOVL C00461 V=20.0 PL=1
MOVL C00462 V=130.0 PL=1
MOVL C00463 V=130.0 PL=1
MOVL C00464 V=60.0 PL=1
MOVL C00465 V=60.0 PL=1
MOVL C00466 V=60.0 PL=1
MOVL C00467 V=60.0 PL=1
MOVL C00468 V=130.0 PL=1
MOVL C00469 V=30.0 PL=1
MOVL C00470 V=30.0 PL=1
MOVL C00471 V=30.0 PL=1
MOVL C00472 V=30.0 PL=1
MOVL C00473 V=30.0 PL=1
MOVL C00474 V=30.0 PL=1
MOVL C00475 V=30.0 PL=1
MOVL C00476 V=30.0 PL=1
MOVL C00477 V=130.0 PL=1
MOVL C00478 V=130.0 PL=1
MOVL C00479 V=20.0 PL=1
MOVL C00480 V=130.0 PL=1
MOVL C00481 V=130.0 PL=1
MOVL C00482 V=60.0 PL=1
MOVL C00483 V=60.0 PL=1
MOVL C00484 V=60.0 PL=1
MOVL C00485 V=60.0 PL=1
MOVL C00486 V=130.0 PL=1
MOVL C00487 V=30.0 PL=1
MOVL C00488 V=30.0 PL=1
MOVL C00489 V=30.0 PL=1
MOVL C00490 V=30.0 PL=1
MOVL C00491 V=30.0 PL=1
MOVL C00492 V=30.0 PL=1
MOVL C00493 V=30.0 PL=1
MOVL C00494 V=30.0 PL=1
MOVL C00495 V=130.0 PL=1
MOVL C00496 V=130.0 PL=1
MOVL C00497 V=20.0 PL=1
MOVL C00498 V=130.0 PL=1
MOVL C00499 V=130.0 PL=1
MOVL C00500 V=60.0 PL=1
MOVL C00501 V=60.0 PL=1
MOVL C00502 V=60.0 PL=1
MOVL C00503 V=60.0 PL=1
MOVL C00504 V=130.0 PL=1
MOVL C00505 V=30.0 PL=1
MOVL C00506 V=30.0 PL=1
MOVL C00507 V=30.0 PL=1
MOVL C00508 V=30.0 PL=1
MOVL C00509 V=30.0 PL=1
MOVL C00510 V=30.0 PL=1
MOVL C00511 V=30.0 PL=1
MOVL C00512 V=30.0 PL=1
MOVL C00513 V=130.0 PL=1
MOVL C00514 V=130.0 PL=1
MOVL C00515 V=20.0 PL=1
MOVL C00516 V=130.0 PL=1
MOVL C00517 V=130.0 PL=1
MOVL C00518 V=60.0 PL=1
MOVL C00519 V=60.0 PL=1
MOVL C00520 V=60.0 PL=1
MOVL C00521 V=60.0 PL=1
MOVL C00522 V=130.0 PL=1
MOVL C00523 V=30.0 PL=1
MOVL C00524 V=30.0 PL=1
MOVL C00525 V=30.0 PL=1
MOVL C00526 V=30.0 PL=1
MOVL C00527 V=30.0 PL=1
MOVL C00528 V=30.0 PL=1
MOVL C00529 V=30.0 PL=1
MOVL C00530 V=30.0 PL=1
MOVL C00531 V=130.0 PL=1
MOVL C00532 V=130.0 PL=1
MOVL C00533 V=20.0 PL=1
MOVL C00534 V=130.0 PL=1
MOVL C00535 V=130.0 PL=1
MOVL C00536 V=60.0 PL=1
MOVL C00537 V=60.0 PL=1
MOVL C00538 V=60.0 PL=1
MOVL C00539 V=60.0 PL=1
MOVL C00540 V=130.0 PL=1
MOVL C00541 V=30.0 PL=1
MOVL C00542 V=30.0 PL=1
MOVL C00543 V=30.0 PL=1
MOVL C00544 V=30.0 PL=1
MOVL C00545 V=30.0 PL=1
MOVL C00546 V=30.0 PL=1
MOVL C00547 V=30.0 PL=1
MOVL C00548 V=30.0 PL=1
MOVL C00549 V=130.0 PL=1
MOVL C00550 V=130.0 PL=1
MOVL C00551 V=20.0 PL=1
MOVL C00552 V=130.0 PL=1
MOVL C00553 V=130.0 PL=1
MOVL C00554 V=60.0 PL=1
MOVL C00555 V=60.0 PL=1
MOVL C00556 V=60.0 PL=1
MOVL C00557 V=60.0 PL=1
MOVL C00558 V=130.0 PL=1
MOVL C00559 V=30.0 PL=1
MOVL C00560 V=30.0 PL=1
MOVL C00561 V=30.0 PL=1
MOVL C00562 V=30.0 PL=1
MOVL C00563 V=30.0 PL=1
MOVL C00564 V=30.0 PL=1
MOVL C00565 V=30.0 PL=1
MOVL C00566 V=30.0 PL=1
MOVL C00567 V=130.0 PL=1
MOVL C00568 V=130.0 PL=1
MOVL C00569 V=20.0 PL=1
MOVL C00570 V=130.0 PL=1
MOVL C00571 V=130.0 PL=1
MOVL C00572 V=60.0 PL=1
MOVL C00573 V=60.0 PL=1
MOVL C00574 V=60.0 PL=1
MOVL C00575 V=60.0 PL=1
MOVL C00576 V=130.0 PL=1
MOVL C00577 V=30.0 PL=1
MOVL C00578 V=30.0 PL=1
MOVL C00579 V=30.0 PL=1
MOVL C00580 V=30.0 PL=1
MOVL C00581 V=30.0 PL=1
MOVL C00582 V=30.0 PL=1
MOVL C00583 V=30.0 PL=1
MOVL C00584 V=30.0 PL=1
MOVL C00585 V=130.0 PL=1
MOVL C00586 V=130.0 PL=1
MOVL C00587 V=20.0 PL=1
MOVL C00588 V=130.0 PL=1
MOVL C00589 V=130.0 PL=1
MOVL C00590 V=60.0 PL=1
MOVL C00591 V=60.0 PL=1
MOVL C00592 V=60.0 PL=1
MOVL C00593 V=60.0 PL=1
MOVL C00594 V=130.0 PL=1
MOVL C00595 V=30.0 PL=1
MOVL C00596 V=30.0 PL=1
MOVL C00597 V=30.0 PL=1
MOVL C00598 V=30.0 PL=1
MOVL C00599 V=30.0 PL=1
MOVL C00600 V=30.0 PL=1
MOVL C00601 V=30.0 PL=1
MOVL C00602 V=30.0 PL=1
MOVL C00603 V=130.0 PL=1
MOVL C00604 V=130.0 PL=1
MOVL C00605 V=20.0 PL=1
MOVL C00606 V=130.0 PL=1
MOVL C00607 V=130.0 PL=1
MOVL C00608 V=60.0 PL=1
MOVL C00609 V=60.0 PL=1
MOVL C00610 V=60.0 PL=1
MOVL C00611 V=60.0 PL=1
MOVL C00612 V=130.0 PL=1
MOVL C00613 V=30.0 PL=1
MOVL C00614 V=30.0 PL=1
MOVL C00615 V=30.0 PL=1
MOVL C00616 V=30.0 PL=1
MOVL C00617 V=30.0 PL=1
MOVL C00618 V=30.0 PL=1
MOVL C00619 V=30.0 PL=1
MOVL C00620 V=30.0 PL=1
MOVL C00621 V=130.0 PL=1
MOVL C00622 V=130.0 PL=1
MOVL C00623 V=20.0 PL=1
MOVL C00624 V=80.0 PL=1
END
